// TIA Portal project "CO321_PumpControl" (V15)

(* hardware
DEVICE "S7-1200 station_1"  S7-1200 Station
   slot 0: "Rack_0"  S7-1200 Rack  Rack  V1.0
   slot 1: "PLC_1"  CPU 1215C DC/DC/DC  6ES7 215-1AG31-0XB0  V3.0
*)

// ===== PLC "PLC_1"  CPU 1215C DC/DC/DC =====

VAR_GLOBAL   // PLC tag table "Default tag table"
   "Reservoir Low" AT %I0.0 : Bool;
   "Reservoir High" AT %I0.1 : Bool;
   "Tank Low" AT %I0.2 : Bool;
   "Tank High" AT %I0.3 : Bool;
   "Pump Manual" AT %I0.4 : Bool;
   "System On" AT %I0.5 : Bool;
   "Pump" AT %Q0.1 : Bool;
   "Valve 01" AT %Q0.0 : Bool;
   "Pump On Light" AT %Q0.2 : Bool;
   "System On Light" AT %Q0.3 : Bool;
   "System Status" AT %M0.0 : Bool;
   "Pump Auto Status" AT %M0.1 : Bool;
   "Pump Manual Status" AT %M0.2 : Bool;
END_VAR

DATA_BLOCK "MB_DB"   // DB1
{ S7_Optimized_Access := 'FALSE' }
VERSION : 0.1
   VAR
      HOLD_REG : Array[0..49] of Word;
      CONNECT : TCON_IP_v4;
      ERROR : Bool;
      STATUS : Word;
      HREG : Struct
         Static_1 : Word;
      END_STRUCT;
   END_VAR
BEGIN
   CONNECT.InterfaceId := 64;
   CONNECT.ID := 1;
   CONNECT.ConnectionType := 11;
   CONNECT.LocalPort := 502;
END_DATA_BLOCK

DATA_BLOCK "modbus"   // DB3
{ S7_Optimized_Access := 'FALSE' }
VERSION : 0.1
   VAR
      data1 : Word := 1;
      data2 : Word := 2;
      data3 : Word := 3;
      data4 : Word := 4;
      data5 : Word := 5;
      data6 : Word := 6;
      data7 : Word := 7;
      data8 : Word := 8;
      data9 : Word;
      data10 : Word;
      data11 : Word;
      data2_1 : Word;
      data3_1 : Word;
      data4_1 : Word;
      data5_1 : Word;
      data6_1 : Word;
      data7_1 : Word;
   END_VAR
BEGIN
END_DATA_BLOCK

ORGANIZATION_BLOCK "Main"   // OB1, LAD, ProgramCycle
TITLE = "Main Program Sweep (Cycle)"
{ S7_Optimized_Access := 'TRUE' }
VERSION : 0.1
BEGIN

REGION Network 1
   // For system status and status light
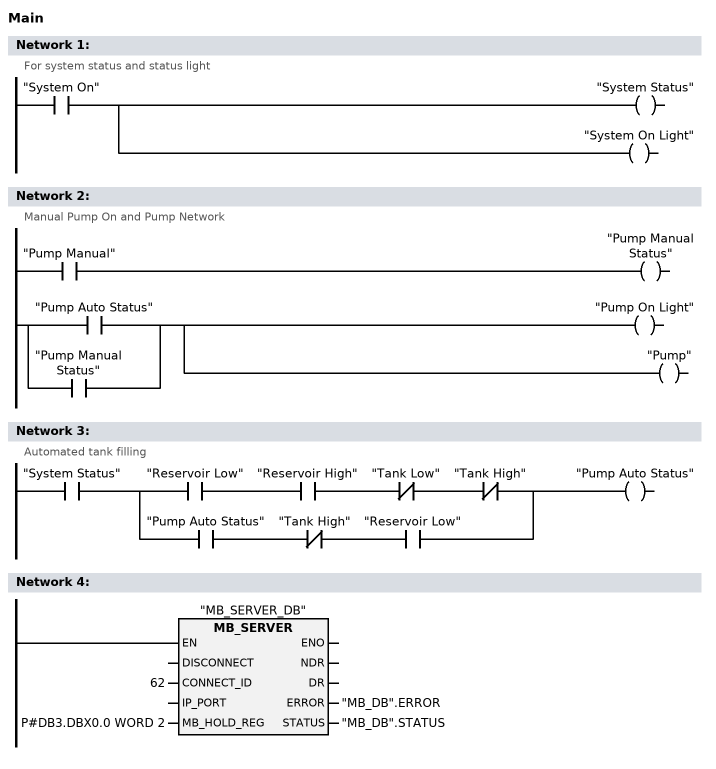
   RUNG wire#powerrail
      Contact( "System On" )
      wire#w1
      Coil( "System Status" )
   END_RUNG
   RUNG wire#w1
      Coil( "System On Light" )
   END_RUNG
   // the same network as SCL:
   "System Status" := "System On";
   "System On Light" := "System On";
END_REGION

REGION Network 2
   // Manual Pump On and Pump Network
   RUNG wire#powerrail
      Contact( "Pump Manual" )
      Coil( "Pump Manual Status" )
   END_RUNG
   RUNG wire#powerrail
      Contact( "Pump Auto Status" )
      wire#w1
      Coil( "Pump On Light" )
   END_RUNG
   RUNG wire#powerrail
      Contact( "Pump Manual Status" )
   END_RUNG wire#w1
   RUNG wire#w1
      Coil( "Pump" )
   END_RUNG
   // the same network as SCL:
   "Pump Manual Status" := "Pump Manual";
   "Pump On Light" := "Pump Auto Status" OR "Pump Manual Status";
   "Pump" := "Pump On Light";
END_REGION

REGION Network 3
   // Automated tank filling
   RUNG wire#powerrail
      Contact( "System Status" )
      wire#w1
      Contact( "Reservoir Low" )
      Contact( "Reservoir High" )
      I_Contact( "Tank Low" )
      I_Contact( "Tank High" )
      wire#w2
      Coil( "Pump Auto Status" )
   END_RUNG
   RUNG wire#w1
      Contact( "Pump Auto Status" )
      I_Contact( "Tank High" )
      Contact( "Reservoir Low" )
   END_RUNG wire#w2
   // the same network as SCL:
   "Pump Auto Status" := "System Status" AND (("Reservoir Low" AND "Reservoir High" AND NOT "Tank Low" AND NOT "Tank High") OR ("Pump Auto Status" AND NOT "Tank High" AND "Reservoir Low"));
END_REGION

REGION Network 4
   "MB_SERVER_DB"(CONNECT_ID := 62,   // MB_SERVER
                  MB_HOLD_REG := P#DB3.DBX0.0 WORD 2,
                  ERROR => "MB_DB".ERROR,
                  STATUS => "MB_DB".STATUS);
END_REGION
END_ORGANIZATION_BLOCK